Fanuc KAREL source: CE0065.KL

PROGRAM CE0065
%STACKSIZE=65535
%PRIORITY=65535
%NOLOCKGROUP
ROUTINE RB(P1 : BOOLEAN) : BOOLEAN FROM CE0065
ROUTINE RI(P1 : INTEGER) : INTEGER FROM CE0065
ROUTINE RR(P1 : REAL) : REAL FROM CE0065
ROUTINE RTEST FROM CE0065
ROUTINE RB
BEGIN
RETURN(P1)
-- UNRESOLVED_PC line 6 opcodes [7F] marker_code=16
END RB
ROUTINE RI
BEGIN
-- UNRESOLVED_PC line 9 opcodes [2D 9D 52 7F] marker_code=26
-- UNRESOLVED_PC line 10 opcodes [7F] marker_code=43
END RI
ROUTINE RR
BEGIN
-- UNRESOLVED_PC line 13 opcodes [2D 2E 69 7F] marker_code=53
-- UNRESOLVED_PC line 14 opcodes [7F] marker_code=74
END RR
ROUTINE RTEST
VAR
L1 : STRING[20]
L2 : STRING[20]
L3 : ARRAY[3] OF INTEGER
S1 : INTEGER
U2C_18 : INTEGER -- ASSUMED 2C source type; see uncertainty report
U2C_19 : INTEGER -- ASSUMED 2C source type; see uncertainty report
U2C_20 : INTEGER -- ASSUMED 2C source type; see uncertainty report
U2C_21 : BOOLEAN -- ASSUMED 2C source type; see uncertainty report
U2C_22 : BOOLEAN -- ASSUMED 2C source type; see uncertainty report
BEGIN
S1=2
U2C_18=3
U2C_19=1075838976
U2C_20=1080033280
U2C_21=TRUE
U2C_22=FALSE
L1='AB'
L2='AC'
L3[1]=2
L3[2]=3
IF (L3[1] > S1) THEN
S1=(S1 + 1)
ELSE
S1=(S1 + 2)
ENDIF
END RTEST
BEGIN
RTEST
END CE0065
